// Mitsubishi GX Works2 project: GT_EX2   PLC: Q03UDV

PROGRAM MAIN
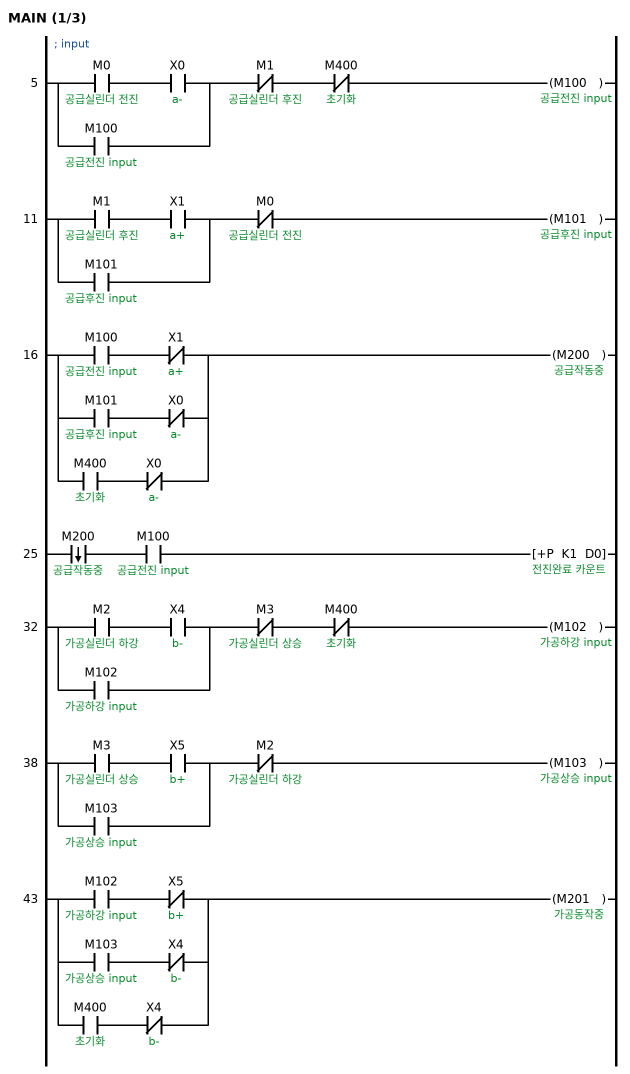
; input
5     LD      M0  ; 공급실린더 전진
      AND     X0  ; a-
      OR      M100  ; 공급전진 input
      ANI     M1  ; 공급실린더 후진
      ANI     M400  ; 초기화
      OUT     M100  ; 공급전진 input
11    LD      M1  ; 공급실린더 후진
      AND     X1  ; a+
      OR      M101  ; 공급후진 input
      ANI     M0  ; 공급실린더 전진
      OUT     M101  ; 공급후진 input
16    LD      M100  ; 공급전진 input
      ANI     X1  ; a+
      LD      M101  ; 공급후진 input
      ANI     X0  ; a-
      ORB
      LD      M400  ; 초기화
      ANI     X0  ; a-
      ORB
      OUT     M200  ; 공급작동중
25    LDF     M200  ; 공급작동중
      AND     M100  ; 공급전진 input
      +P      K1 D0  ; 전진완료 카운트
32    LD      M2  ; 가공실린더 하강
      AND     X4  ; b-
      OR      M102  ; 가공하강 input
      ANI     M3  ; 가공실린더 상승
      ANI     M400  ; 초기화
      OUT     M102  ; 가공하강 input
38    LD      M3  ; 가공실린더 상승
      AND     X5  ; b+
      OR      M103  ; 가공상승 input
      ANI     M2  ; 가공실린더 하강
      OUT     M103  ; 가공상승 input
43    LD      M102  ; 가공하강 input
      ANI     X5  ; b+
      LD      M103  ; 가공상승 input
      ANI     X4  ; b-
      ORB
      LD      M400  ; 초기화
      ANI     X4  ; b-
      ORB
      OUT     M201  ; 가공동작중
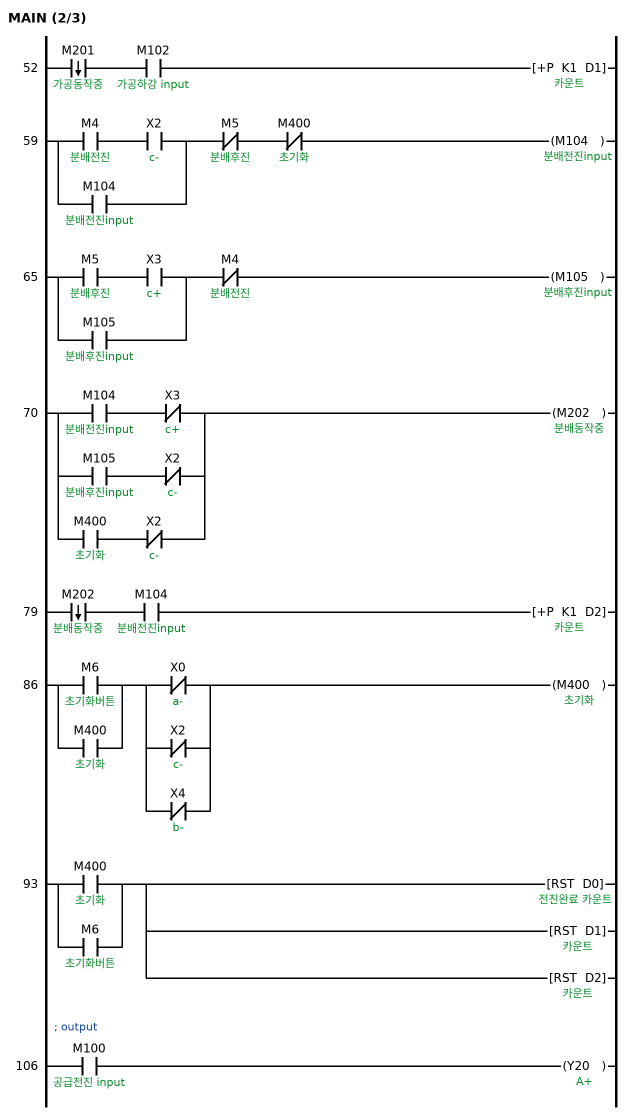
52    LDF     M201  ; 가공동작중
      AND     M102  ; 가공하강 input
      +P      K1 D1  ; 카운트
59    LD      M4  ; 분배전진
      AND     X2  ; c-
      OR      M104  ; 분배전진input
      ANI     M5  ; 분배후진
      ANI     M400  ; 초기화
      OUT     M104  ; 분배전진input
65    LD      M5  ; 분배후진
      AND     X3  ; c+
      OR      M105  ; 분배후진input
      ANI     M4  ; 분배전진
      OUT     M105  ; 분배후진input
70    LD      M104  ; 분배전진input
      ANI     X3  ; c+
      LD      M105  ; 분배후진input
      ANI     X2  ; c-
      ORB
      LD      M400  ; 초기화
      ANI     X2  ; c-
      ORB
      OUT     M202  ; 분배동작중
79    LDF     M202  ; 분배동작중
      AND     M104  ; 분배전진input
      +P      K1 D2  ; 카운트
86    LD      M6  ; 초기화버튼
      OR      M400  ; 초기화
      LDI     X0  ; a-
      ORI     X2  ; c-
      ORI     X4  ; b-
      ANB
      OUT     M400  ; 초기화
93    LD      M400  ; 초기화
      OR      M6  ; 초기화버튼
      RST     D0  ; 전진완료 카운트
      RST     D1  ; 카운트
      RST     D2  ; 카운트
; output
106   LD      M100  ; 공급전진 input
      OUT     Y20  ; A+
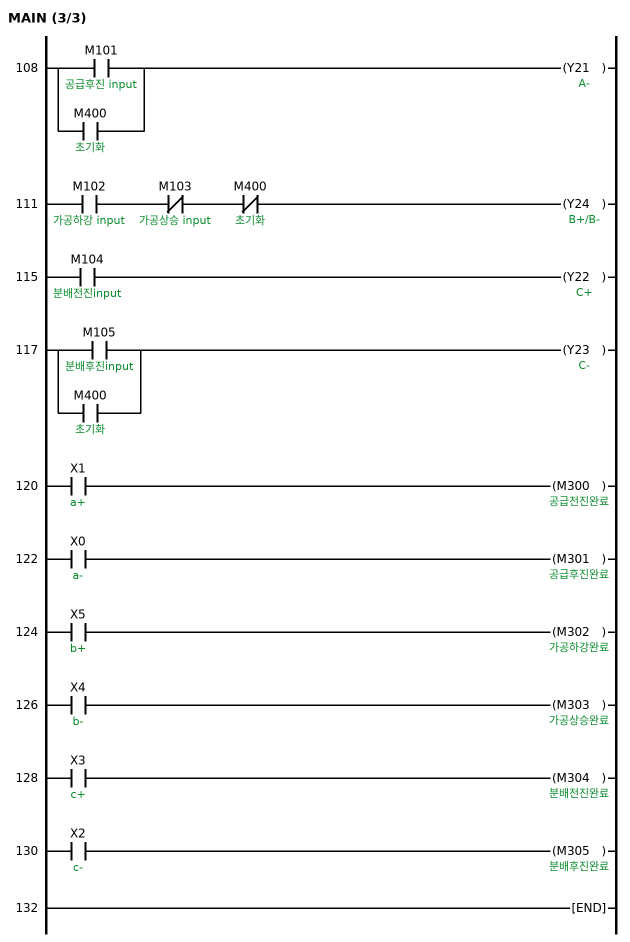
108   LD      M101  ; 공급후진 input
      OR      M400  ; 초기화
      OUT     Y21  ; A-
111   LD      M102  ; 가공하강 input
      ANI     M103  ; 가공상승 input
      ANI     M400  ; 초기화
      OUT     Y24  ; B+/B-
115   LD      M104  ; 분배전진input
      OUT     Y22  ; C+
117   LD      M105  ; 분배후진input
      OR      M400  ; 초기화
      OUT     Y23  ; C-
120   LD      X1  ; a+
      OUT     M300  ; 공급전진완료
122   LD      X0  ; a-
      OUT     M301  ; 공급후진완료
124   LD      X5  ; b+
      OUT     M302  ; 가공하강완료
126   LD      X4  ; b-
      OUT     M303  ; 가공상승완료
128   LD      X3  ; c+
      OUT     M304  ; 분배전진완료
130   LD      X2  ; c-
      OUT     M305  ; 분배후진완료
132   END
END_PROGRAM
